ABB RobotStudio station: EstacionTaladrado_20230515-193437.rsstn

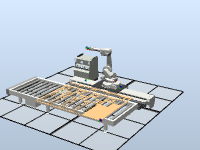
Station EstacionTaladrado (saved by RobotStudio 6.8.8307.1040)
Controller IRB1600APM, task T_ROB1: task frame (RAPID world) sits at (108, -475.5, 460) mm, rotated rx 0 ry 0 rz 90 deg in the station
Controller IRB1600APM
  mechanical unit ROB_1: IRB1600_6_145__02_5, 6 joints, base frame (0, 0, 0) mm
  mechanical unit TRACK_1: IRBT2005_IRB_STD_INT_0_0_3__01, 1 joints, base frame (0, 0, 0) mm
Layout (positions relative to the parent item):
  - Placa_de_Corte [part] at (-2250, -1220, 450) mm
  - IRC5_Singel-Cabinet [part, from Equipment\IRC5_Singel-Cabinet.rslib] at (1200, 1600, 100) mm, rotated rx 90 ry 0 rz 90 deg
  - 1320_4000_h2 [part, from Equipment\Conveyor 1320 4000 h2.rslib] at (-1985, 2600, 0) mm, rotated rx 0 ry 0 rz -90 deg
  - IRB1600_6_145__02_5 [mechanism, from Robots\IRB1600_6_145_G_02.rslib] at (108, -50.5, 460) mm, rotated rx 0 ry 0 rz 90 deg; joint values [0, 0, 0, 0, 0, 0] (rad or m)
  - IRBT2005_IRB_STD_INT_0_0_3__01 [mechanism] at (400, -1300, 0) mm, rotated rx 0 ry 0 rz 90 deg; joint values [0.425] (rad or m)
      links: Base, Link1
  - Ventosa_Smart [smart component]
      signals: DI StartAttacher, DO Executed
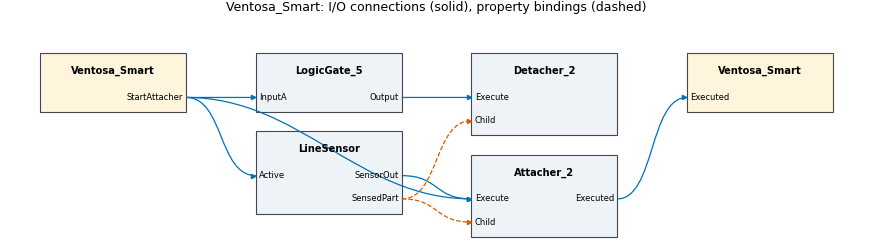
      connections:
        Ventosa_Smart.StartAttacher -> LogicGate_5.InputA
        LogicGate_5.Output -> Detacher_2.Execute
        Ventosa_Smart.StartAttacher -> LineSensor.Active
        LineSensor.SensorOut -> Attacher_2.Execute
        Ventosa_Smart.StartAttacher -> Attacher_2.Execute
        Attacher_2.Executed -> Ventosa_Smart.Executed
        LineSensor.SensedPart => Attacher_2.Child
        LineSensor.SensedPart => Detacher_2.Child
    - Attacher_2 [smart component, from Components\Attacher.rslib]
        properties: Parent=Ventosa; Flange=0; Child=PLACA_SOPORTE_1; Mount=false; Offset=[0 0 0]; Orientation=[0 0 0]
    - Detacher_2 [smart component, from Components\Detacher.rslib]
        properties: Child=PLACA_SOPORTE_1; KeepPosition=true
    - LogicGate_5 [smart component, from Components\LogicGate.rslib]
        properties: Operator=NOT; Delay=0
    - LineSensor [smart component, from Components\LineSensor.rslib] at (108, 874.5, 1646.5) mm, rotated rx 0 ry 90 rz 90 deg
        properties: Start=[0 0 0]; End=[6.66133814775094E-16 -4.71844785465692E-16 0.00999998807907376]; Radius=0.001; SensedPart=PLACA_SOPORTE_1; SensedPoint=[-1.19998193359375 0.989787048339844 0.462]
      - _sensorPart_ [part]
    - Ventosa [mechanism, from Libraries\Ventosa.rslib] at (108, 764.5, 1646.5) mm, rotated rx 0 ry 90 rz 90 deg
  - PLACA_SOPORTE_1 [part] at (-1200.46, 988.98, 450) mm
Attachment: IRB1600_6_145__02_5 is attached to IRBT2005_IRB_STD_INT_0_0_3__01 / Link1
Attachment: Ventosa is attached to IRB1600_6_145__02_5 / Link6
Attachment: LineSensor is attached to Ventosa / HERRAMIENTA
Station logic (signal -> signal, property => property):
  Attacher.Executed -> LogicGate.InputB
  IRB1600APM.DOATTCH -> Ventosa_Smart.StartAttacher
Targets, tools, work objects and paths stored in the station, written as RAPID:
! task T_ROB1
MODULE CalibData
  PERS tooldata VentosaTCP:=[TRUE,[[0,0,110.772],[1,0,0,0]],[1,[0,0,53.582],[1,0,0,0],0,0,0]];
  TASK PERS wobjdata Placa:=[FALSE,TRUE,"",[[0,0,0],[1,0,0,0]],[[-744.5,2358,-10],[0.707106781,0,0,-0.707106781]]];
ENDMODULE

! task T_ROB1
MODULE Module1
  CONST jointtarget MID_POINT:=[[90,70,-70,0,90,0],[425,9E+09,9E+09,9E+09,9E+09,9E+09]];
  CONST robtarget PLACA_SOPORTE_1:=[[1050.01804282,2209.787180675,12.000031193],[-0.000000003,0.999795002,-0.020247298,0.000000052],[0,-1,-1,0],[1350,9E+09,9E+09,9E+09,9E+09,9E+09]];
  CONST jointtarget HOME:=[[0,0,0,0,0,0],[425,9E+09,9E+09,9E+09,9E+09,9E+09]];
  PROC Path_MID_POINT()
    MoveAbsJ MID_POINT,v1000,z100,VentosaTCP\WObj:=Placa;
  ENDPROC
  PROC Path_PLACA_SOPORTE_1()
    MoveJ PLACA_SOPORTE_1,v1000,z100,VentosaTCP\WObj:=Placa;
  ENDPROC
  PROC Path_HOME()
    MoveAbsJ HOME,v1000,z100,VentosaTCP\WObj:=Placa;
  ENDPROC
  PROC main()
    Path_HOME;
    Path_MID_POINT;
    Path_PLACA_SOPORTE_1;
    WaitDO DOATTCH,1;
    Path_MID_POINT;
    Path_PLACA_SOPORTE_1;
    WaitDO DOATTCH,0;
    Path_MID_POINT;
    Path_HOME;
  ENDPROC
ENDMODULE

